// TIA Portal V20 export
TYPE "LKinCtrl_typePathDataElement_reduced"
   STRUCT
      cmdType : Int := -1;   // 1: MoveLinAbs; 2: MoveLinRel; 100: WaitTime; 0: FlagOnlyCmd; -1: End of List
      cmdActivated : Bool := TRUE;   // (de)activation of command
      cmdName : String["LKINCTRL_LENGTH_OF_CMDPOINT_NAME"];   // name of command
      point : DInt := -1;   // reference to point table, used for cmdCoordinates
      cmdCoordinates : "LKinCtrl_typePointCoordinates";   // target coordinate definition
      cmdParameters : "LKinCtrl_typePointParameter_reduced";   // additional command parameters
      setFlags : Array[1.."LKINCTRL_NO_OF_CMD_SETFLAGS"] of "LKinCtrl_typeSetFlagElement_Bool";   // flags to control actuators
      valueFlags : Array[1.."LKINCTRL_NO_OF_CMD_VALUEFLAGS"] of "LKinCtrl_typeSetFlagElement_LReal";   // value flags to control actuators
   END_STRUCT;
   // cmdParameters.transitionParameters[1] := -1.0;
END_TYPE
